{attribute 'GeneratedUsingTerminal: EL6224-0090-0016'}
{attribute addProperty BoxType "EL6224-0090-0016"}
{attribute addProperty Id "DeviceState_InputsDeviceState_Inputs_4751FF764"}
{attribute addProperty CRC "3178000437"}
{attribute addProperty Size "4"}
TYPE Module_2_DeviceState_Inputs_BD6C7035 :
STRUCT
	{attribute addProperty Name "DeviceState_Inputs"}
	DeviceState_Inputs  : DeviceState_Inputs_4751FF76;
END_STRUCT
END_TYPE

(* stored: Version 1.2.0.0, ProductVersion 3.1.4024.11
   DUT Module_2_DeviceState_Inputs_BD6C7035: Id {efd0e6c8-609c-4e17-b33e-2746460ab9dc} *)
